(* IEC 61131-3 sources: Industry-PLC-LLM/data/PLCBEAD_repo/PLCBEAD_PLCEmbed-main/PLC-BEAD/Source/GEB/ISC_CTRL, 1 file *)

(* ---- ISC_CTRL.ST ---- *)
FUNCTION ISC_CTRL:BOOL

	VAR_INPUT
		IN :	BYTE;
	END_VAR

	ISC_CTRL := IN < BYTE#32 OR IN = BYTE#127;

END_FUNCTION

PROGRAM program0
	VAR
		IN : BYTE;
		OUT : BOOL;
	END_VAR

	OUT := ISC_CTRL(IN);
END_PROGRAM
